(* IEC 61131-3 sources: brOscatLib/oscatBuild, 60 files *)

(* ---- oscatBuild.typ ---- *)
TYPE
END_TYPE

(* ---- AIR_DENSITY.st ---- *)
FUNCTION AIR_DENSITY
    (*http://www.oscat.de/images/OSCATBasic/oscat_basic333_en.pdf#page=426*)
    AIR_DENSITY := cPN * (1.0 - RH * SDD(T, TRUE) * RX / P) / (RL * ( T - cT0));

    (* original code used for rev 1.0

    SDD := SDD(T,FALSE);
    RF := RL / (1- RH*SDD/P*RX);
    AIR_DENSITY := P / (RF * (T-TK));

    *)

    (* revision history

    hm	29.10.2007	rev 1.0
    	original version

    hm	4.12.2007		rev 1.1
    	changed code for better performance

    hm	18. oct. 2008	rev 1.2
    	using phys constants

    hm	13. mar. 2009	rev 1.3
    	real constants updated to new systax using dot

    *)

END_FUNCTION

(* ---- AIR_ENTHALPY.st ---- *)
FUNCTION AIR_ENTHALPY
    (*http://www.oscat.de/images/OSCATBasic/oscat_basic333_en.pdf#page=427*)
    AIR_ENTHALPY := CPL * T + (CW * T + LH) * DEW_CON(RH,T);

    (* revision history

    hm	31.10.2007	rev 1.0
    	original version

    hm	2.11.2007		rev 1.1
    	deleted unused variable RF

    hm	2.12.2007		rev 1.2
    	changed code for better performance
    *)

END_FUNCTION

(* ---- BUILDING_VERSION.st ---- *)
FUNCTION BUILDING_VERSION
    (*http://www.oscat.de/images/OSCATBuilding/oscat_building100_en.pdf#page=11*)
    IF IN THEN
    	BUILDING_VERSION := DATE_TO_DWORD(D#2011-02-3);
    ELSE
    	BUILDING_VERSION := 100;
    END_IF

    (* revision history
    hm	6. oct 2006	rev 1.0
    	original version

    hm	16. dec 2007	rev 1.1
    	added possibility to return date and version depending on IN.

    *)
END_FUNCTION

(* ---- DEW_CON.st ---- *)
FUNCTION DEW_CON
    (*http://www.oscat.de/images/OSCATBasic/oscat_basic333_en.pdf#page=434*)
    (*	this code is good to read but need to be improoved
    	SDD := 6.1078*EXPT(10,(a*T)/(b+T));
    	DD := RH/100 * SDD;
    	V := LOG(DD/6.1078);
    	TD := b*V/(a-v);
    	DEW_CON := 0.1 * mw / RU * DD / (T - TK);
    *)
    IF RH > 0.0 AND T > -50.0 THEN
    	DEW_CON := 2.166824303E-2 * RH * SDD(T,FALSE)  / (T - cT0);
    ELSE
    	DEW_CON := 0.0;
    END_IF

    (*
    Bezeichnungen:
    r = relative Luftfeuchte
    T = Temperatur in °C
    TK = Temperatur in Kelvin (TK = T + 273.15)
    TD = Taupunkttemperatur in °C
    DD = Dampfdruck in hPa
    SDD = Sättigungsdampfdruck in hPa

    Parameter:
    a = 7.5, b = 237.3 für T >= 0
    a = 7.6, b = 240.7 für T < 0 über Wasser (Taupunkt)
    a = 9.5, b = 265.5 für T < 0 über Eis (Frostpunkt)

    R* = 8314.3 J/(kmol*K) (universelle Gaskonstante)
    mw = 18.016 kg (Molekulargewicht des Wasserdampfes)
    AF = absolute Feuchte in g Wasserdampf pro m3 Luft

    Formeln:

       1. SDD(T) = 6.1078 * 10((a*T)/(b+T))
       2. DD(r,T) = r/100 * SDD(T)
       3. r(T,TD) = 100 * SDD(TD) / SDD(T)
       4. TD(r,T) = b*v/(a-v) mit v(r,T) = log10(DD(r,T)/6.1078)
       5. AF(r,TK) = 105 * mw/R* * DD(r,T)/TK; AF(TD,TK) = 105 * mw/R* * SDD(TD)/TK

    *)

    (* revision history

    hm 29 apr 2007	rev 1.0
    	original version

    hm	13.sep 2007	rev 1.1
    	improoved coding for speed
    	deleted unused variabled SDD,DD,V, TD

    hm	2. dec 2007	rev 1.2
    	changed code for better performance
    	output is now in Gramms / Qubic meter

    hm	14. oct. 2008	rev 1.3
    	performance improvement

    hm	18. oct. 2008	rev 1.4
    	using phys constants

    hm	13. mar. 2009	rev 1.5
    	improved code

    hm	19. jan. 2011	rev 1.6
    	return value 0.0 if RH <= 0.0

    *)
END_FUNCTION

(* ---- DEW_RH.st ---- *)
FUNCTION DEW_RH
    (*http://www.oscat.de/images/OSCATBasic/oscat_basic333_en.pdf#page=435*)
    DEW_RH := LIMIT(0.0, VC / DEW_CON(1.0, T), 100.0);

    (* code before rev 1.1
    DEW_RH := VC / dew_con(100,T) * 100;
    IF DEW_RH > 100 THEN DEW_RH := 100; END_IF
    *)

    (* revision history
    hm	29. apr 2007	rev 1.0
    	original version

    hm	2. 12. 2007	rev 1.1
    	new code for better performance

    hm	13. mar. 2009	rev 1.2
    	real constants updated to new systax using dot

    *)
END_FUNCTION

(* ---- DEW_TEMP.st ---- *)
FUNCTION DEW_TEMP
    (*http://www.oscat.de/images/OSCATBasic/oscat_basic333_en.pdf#page=436*)
    IF RH > 0.0 THEN
    (*	old code was rewritten for better performance
    	SDD := 6.1078*EXPT(10,(a*T)/(b+T));
    	DD := RH/100 * SDD;
    	V := LOG(DD/6.1078);
    	DEW_TEMP := b*V/(a-V);
    *)
    	V := LOG(RH * 0.01 * EXP10((a*T) / (b+T)));
    	DEW_TEMP := b*V / (a-V);
    ELSE
    	DEW_TEMP:= cT0;
    END_IF

    (* revision history

    hm		2.10.2006	rev 1.0
    	original version created

    hm		29.4.2007	rev 1.1
    	checked for RH not to be 0 because log(0) is not defined

    hm		13.9.2007	rev 1.2
    	code rewritten for better performance

    hm	2. dec 2007	rev 1.3
    	changed code for better performance

    hm	8. jan 2008	rev 1.4
    	further improvement in performance

    hm	18. oct. 2008	rev 1.5
    	using phys constants

    hm	13. mar. 2009	rev 1.6
    	real constants updated to new systax using dot
    	function will now return -273.15 °C for RH = 0
    *)

    (*
    Bezeichnungen:
    r = relative Luftfeuchte
    T = Temperatur in °C
    TK = Temperatur in Kelvin (TK = T + 273.15)
    TD = Taupunkttemperatur in °C
    DD = Dampfdruck in hPa
    SDD = Sättigungsdampfdruck in hPa

    Parameter:
    a = 7.5, b = 237.3 für T >= 0
    a = 7.6, b = 240.7 für T < 0 über Wasser (Taupunkt)
    a = 9.5, b = 265.5 für T < 0 über Eis (Frostpunkt)

    R* = 8314.3 J/(kmol*K) (universelle Gaskonstante)
    mw = 18.016 kg (Molekulargewicht des Wasserdampfes)
    AF = absolute Feuchte in g Wasserdampf pro m3 Luft

    Formeln:

       1. SDD(T) = 6.1078 * 10((a*T)/(b+T))
       2. DD(r,T) = r/100 * SDD(T)
       3. r(T,TD) = 100 * SDD(TD) / SDD(T)
       4. TD(r,T) = b*V/(a-V) mit V(r,T) = log10(DD(r,T)/6.1078)
       5. AF(r,TK) = 105 * mw/R* * DD(r,T)/TK; AF(TD,TK) = 105 * mw/R* * SDD(TD)/TK

    *)
END_FUNCTION

(* ---- HEAT_INDEX.st ---- *)
FUNCTION HEAT_INDEX
    (*http://www.oscat.de/images/OSCATBasic/oscat_basic333_en.pdf#page=436*)
    IF RH < 20.0 OR T < 20.0 THEN
    	HEAT_INDEX := T;
    ELSE
    	RH2 := RH * RH;
    	T := C_TO_F(T);
    	T2 := T * T;
    	HEAT_INDEX := -42.379 + 2.04901523 * T - 6.83783E-3 * T2
    			+ RH * (10.1433127 - 0.22475541 * T + 1.22874E-3 * T2)
    			+ RH2 * (8.5282E-4 * T - 5.481717E-2 - 1.99E-6 * T2);
    	HEAT_INDEX := F_TO_C(HEAT_INDEX);
    END_IF

    (* revision history

    hm 27.2.2007		rev 1.1
    	deleted unused variables rh3 and T3

    hm	2.12.2007		rev 1.2
    	changed code for better performance

    hm	13. mar. 2009	rev 1.3
    	real constants updated to new systax using dot

    *)
END_FUNCTION

(* ---- SDD.st ---- *)
FUNCTION SDD
    (*http://www.oscat.de/images/OSCATBasic/oscat_basic333_en.pdf#page=445*)
    IF ICE THEN
    	SDD := 611.153 * EXP(22.4433 * T / (272.186 + T));
    ELSE
    	SDD := 611.213 * EXP(17.5043 * T / (241.2 + T));
    END_IF

    (* revision history

    hm 29 oct 2007		rev 1.0
    	original version

    hm	2. dec 2007		rev 1.1
    	changed code for better performance
    *)
END_FUNCTION

(* ---- SDD_NH3.st ---- *)
FUNCTION SDD_NH3
    (*http://www.oscat.de/images/OSCATBasic/oscat_basic333_en.pdf#page=446*)
    (*
    calculate according to NIST
    Antoine Equation Parameters
    log10(P) = A - (B / (T + C))
    	P = vapor pressure (bar)
    	T = temperature (K)
    Temperature (K)	A	B	C	Reference	Comment

     T = 164.0 - 239.5, A =	3.18757, B =506.713, C=-80.78	Stull, 1947	Coefficents calculated by NIST from author's data.
     T = 239.5 - 371.4, A =	4.86886, B = 1113.928, C = -10.409	Stull, 1947	Coefficents calculated by NIST from author's data.
    *)

    IF T < -33.65 THEN
    	SDD_NH3 := EXP(7.3396511649 - ( 1166.7498002 / ( T + 192.37 )));
    ELSE
    	SDD_NH3 := EXP(11.210964456 - ( 2564.9140075 / ( T + 262.741 )));
    END_IF

    (* revision history

    hm 19 aug 2009		rev 1.0
    	original version

    *)
END_FUNCTION

(* ---- SDT_NH3.st ---- *)
FUNCTION SDT_NH3
    (*http://www.oscat.de/images/OSCATBasic/oscat_basic333_en.pdf#page=446*)
    (*
    calculate according to NIST
    Antoine Equation Parameters
    log10(P) = A - (B / (T + C))
    	P = vapor pressure (bar)
    	T = temperature (K)
    Temperature (K)	A	B	C	Reference	Comment

     T = 164.0 - 239.5, A =	3.18757, B =506.713, C=-80.78	Stull, 1947	Coefficents calculated by NIST from author's data.
     T = 239.5 - 371.4, A =	4.86886, B = 1113.928, C = -10.409	Stull, 1947	Coefficents calculated by NIST from author's data.
    *)

    IF P < 1.0E-3 THEN
    	SDT_NH3 := -110.0;
    ELSIF P < 1.0 THEN
    	SDT_NH3 := 506.713 / (3.18757 - LOG(P)) - 192.37 ;
    ELSE
    	SDT_NH3 := 1113.928 / (4.86886 - LOG(P)) - 262.71 ;
    END_IF

    (* revision history

    hm 20 aug 2009		rev 1.0
    	original version

    *)
END_FUNCTION

(* ---- TANK_VOL1.st ---- *)
FUNCTION TANK_VOL1
    (*http://www.oscat.de/images/OSCATBasic/oscat_basic333_en.pdf#page=448*)
    TANK_VOL1 := CIRCLE_SEG(TR, H) * TL;

    (* revision histroy
    hm	10. mar 2010	rev 1.0
    	original version

    *)
END_FUNCTION

(* ---- TANK_VOL2.st ---- *)
FUNCTION TANK_VOL2
    (*http://www.oscat.de/images/OSCATBasic/oscat_basic333_en.pdf#page=448*)
    TANK_VOL2 := cPI * H * H * (TR - H/3.0);

    (* revision histroy
    hm	10. mar 2010	rev 1.0
    	original version

    *)
END_FUNCTION

(* ---- TIMER_EVENT_DECODE.st ---- *)
FUNCTION TIMER_EVENT_DECODE
    (*http://www.oscat.de/images/OSCATBuilding/oscat_building100_en.pdf#page=62*)
    (* a timer EVENT is specified as follows:
    	$typ;ch;day;start;duration;land;lor#
    $ 		= start of definition
    typ 	= type of definition	(number)
    channel	= channel number		(number)
    day 	= day number			(number)
    start	= start time			(time of day)
    duration= duration of EVENT		(time)
    land	= mask for output AND	(8bit value)
    lor		= mask for ourput OR	(8bit value)
    #		= end of definition
    *)

    (* check for start and ending character *)
    IF (LEFT(EVENT,1) <> '<') AND (RIGHT(EVENT,1) <> '>') THEN RETURN; END_IF
    stop := LEN(EVENT);
    pt := ADR(EVENT);
    start := 2;

    (* parse the string for next ; *)
    FOR pos := 2 TO stop DO
    	IF pt[pos] = 59 OR pt[pos] = 62 THEN
    		tmp := MID(EVENT, pos - start, start);
    		CASE step OF
    			0:	(* read type *)
    				TIMER_EVENT_DECODE.typ := FSTRING_TO_BYTE(tmp);

    			1:	(* read channel *)
    				TIMER_EVENT_DECODE.channel := FSTRING_TO_BYTE(tmp);

    			2:	(* read day *)
    				IF IS_CC(tmp,'0123456789abcdefABCDEF#') THEN
    					TIMER_EVENT_DECODE.day := FSTRING_TO_BYTE(tmp);
    				ELSIF TIMER_EVENT_DECODE.typ = 2 THEN
    					TIMER_EVENT_DECODE.DAY := FSTRING_TO_WEEK(tmp, LANG);
    				ELSE
    					TIMER_EVENT_DECODE.DAY := INT_TO_BYTE(FSTRING_TO_WEEKDAY(tmp, LANG));
    				END_IF

    			3:	(* read start *)
    				TIMER_EVENT_DECODE.start := STRING_TO_TOD(tmp);

    			4:	(* read duaration *)
    				TIMER_EVENT_DECODE.duration := STRING_TO_TIME(tmp);

    			5:	(* read land *)
    				TIMER_EVENT_DECODE.land := FSTRING_TO_BYTE(tmp);

    			6:	(* read lor *)
    				TIMER_EVENT_DECODE.LOR := FSTRING_TO_BYTE(tmp);
    		END_CASE
    		start := pos + 1;
    		step := step + 1;
    	END_IF
    END_FOR

    (* revision history
    hm	17. jun 2008	rev 1.0
    	original version

    hm	25. oct. 2008	rev 1.1
    	adding input LANG for language selection
    *)

END_FUNCTION

(* ---- WATER_CP.st ---- *)
FUNCTION WATER_CP
    (*http://www.oscat.de/images/OSCATBasic/oscat_basic333_en.pdf#page=452*)
    WATER_CP := LINEAR_INT(T, data, Pts);

    (*
        °C - die Celsius-Temperatur in Grad Celsius
        v – das spezifische Volumen in Kubikdezimeter je Kilogramm dm³/kg
        h – die spezifische Enthalpie in Kilojoule je Kilogramm 	kJ/kg
        u – die spezifische Innere Energie in Kilojoule je Kilogramm 	kJ/kg
        s – die spezifische Entropie in Kilojoule je Kilogramm mal Kelvin 	kJ/(kg·K)
        cp - die spezifische Wärmekapazität bei konstantem Druck in Kilojoule je Kilogramm mal Kelvin 	kJ/(kg·K)
        Y – Volumenausdehnungskoeffizient in 10-3 durch Kelvin  10-3/K
        L – Wärmeleitfähigkeit in Milliwatt je Meter mal Kelvin  mW / (m·K)
        n – Viskosität in Mikropascal mal Sekunde uPa·s
        s ? – Oberflächenspannung in Millinewton je Meter  mN/m

    °C 		v 				h 			u 		s 			cp 		Y 		L		n		s
    -20		1,006580
    0 		1,000160 		0,06 		-0,04 	-0,0001 	4,228 	-0,080 	561,0 	1792 	75,65
    4		1,000028
    5 		1,0000 		21,1 		21,0 	0,076 		4,200 	0,011 	570,6 	1518 	74,95
    10 		1,0003 		42,1 		42,0 	0,151 		4,188 	0,087 	580,0 	1306 	74,22
    15 		1,0009 		63,0 		62,9 	0,224 		4,184 	0,152 	589,4 	1137 	73,49
    20 		1,001797 		83,9 		83,8 	0,296 		4,183 	0,209 	598,4 	1001 	72,74
    25 		1,0029 		104,8 		104,7 	0,367 		4,183 	0,259 	607,2 	890,4 	71,98
    30 		1,0044 		125,8 		125,7 	0,437 		4,183 	0,305 	615,5 	797,7 	71,20
    35 		1,0060 		146,7 		146,6 	0,505 		4,183 	0,347 	623,3 	719,6 	70,41
    40 		1,007842 		167,58 	167,5 	0,572 		4,182 	0,386 	630,6 	653,3 	69,60
    45 		1,0099 		188,5 		188,4 	0,638 		4,182 	0,423 	637,3 	596,3 	68,78
    50 		1,0121 		209,4 		209,3 	0,704 		4,181 	0,457 	643,6 	547,1 	67,95
    60 		1,017089 		251,2 		251,1 	0,831 		4,183 	0,522 	654,4 	466,6 	66,24
    70 		1,0227 		293,1 		293,0 	0,955 		4,187 	0,583 	663,1 	404,1 	64,49
    80 		1,029027 		335,0 		334,9 	1,075 		4,194 	0,640 	670,0 	354,5 	62,68
    90 		1,0359 		377,0 		376,9 	1,193 		4,204 	0,696 	675,3 	314,6 	60,82
    99,63 	1,0431 		417,5 		417,4 	1,303 		4,217 	0,748 	679,0 	283,0 	58,99
    100	1,043453		419,1

    Stoffdaten von Wasser Quelle Wickipedia

    Wasser hat unter Normaldruck seine größte Dichte von 1000 Kilogramm pro Kubikmeter bei 3,98 °C und zeigt damit eine Dichteanomalie.
    Diese besteht darin, dass sich Wasser unterhalb von 3,98 °C bei weiterer Temperaturverringerung, auch beim Wechsel zum festen
    Aggregatzustand, wieder ausdehnt, was man nur von wenigen Stoffen kennt. Die derzeit genauesten publizierten Werte für die maximale
    Dichte liegen bei (999,974950 ± 0,00084) kg/m³ und bei (3,983 ± 0,00067) °C für die Temperatur, bei der dieser Wert erreicht wird.
    Die Werte stellen einen Mittelwert der von verschiedenen physikalischen Instituten veröffentlichten Zahlen dar (Stand 2001).

    Die Berechnung der Dichte von luftfreiem Wasser DLF in Abhängigkeit von der Temperatur T ([T] = °C) kann mit Hilfe der folgenden
    Virialgleichung erfolgen:
    : \frac{D_{\rm LF}}{\rm g/l} = \frac{a_0 + a_1 T + a_2 T2 + a_3 T3 + a_4 T4 + a_5 T5}{1 + b T}.
    mit den Koeffizienten: a0 = 999,83952; a1 = 16,952577 (°C)-1; a2 = -7,9905127·10-3 (°C)-2; a3 = -4,6241757·10-5 (°C)-3;
    a4 = 1,0584601·10-7 (°C)-4; a5 = -2,8103006·10-10 (°C)-5 und b = 0,0168872.
    Für die Berechnung der Dichte von luftgesättigtem Wasser korrigiert man den Wert nach
    DLG/(g/l) = DLF/(g/l) - 0,004612 + 0,000106 (°C)-1·T. (Quelle: PTB-Mitteilungen 100/3-90)

    *)

    (* revision history

    hm	29.10.2007	rev 1.0
    	original version

    hm	27. dec 2007	rev 1.1
    	increased accuracy

    hm	13. mar. 2009	rev 1.2
    	real constants updated to new systax using dot

    *)

END_FUNCTION

(* ---- WATER_DENSITY.st ---- *)
FUNCTION WATER_DENSITY
    (*http://www.oscat.de/images/OSCATBasic/oscat_basic333_en.pdf#page=452*)
    T2 := T * T;
    T4 := T2 * T2;
    WATER_DENSITY := (a0 + a1*T + a2*T2 + a3*T2*T + a4*T4 + a5*T4*T) / (1.0 + b*T);
    IF SAT THEN WATER_DENSITY := WATER_DENSITY - 0.004612 + 0.000106 * T; END_IF

    (* revision history

    hm	13.9.2007		rev 1.0
    	original version

    hm	2.12.2007		rev 1.1
    	changed code for better performance

    hm	13. mar. 2009	rev 1.2
    	real constants updated to new systax using dot

    *)

    (*
        °C - die Celsius-Temperatur in Grad Celsius
        v – das spezifische Volumen in Kubikdezimeter je Kilogramm dm³/kg
        h – die spezifische Enthalpie in Kilojoule je Kilogramm 	kJ/kg
        u – die spezifische Innere Energie in Kilojoule je Kilogramm 	kJ/kg
        s – die spezifische Entropie in Kilojoule je Kilogramm mal Kelvin 	kJ/(kg·K)
        cp - die spezifische Wärmekapazität bei konstantem Druck in Kilojoule je Kilogramm mal Kelvin 	kJ/(kg·K)
        Y – Volumenausdehnungskoeffizient in 10-3 durch Kelvin  10-3/K
        L – Wärmeleitfähigkeit in Milliwatt je Meter mal Kelvin  mW / (m·K)
        n – Viskosität in Mikropascal mal Sekunde uPa·s
        s ? – Oberflächenspannung in Millinewton je Meter  mN/m

    °C 		v 				h 			u 		s 			cp 		Y 		L		n		s
    -20		1,006580
    0 		1,000160 		0,06 		-0,04 	-0,0001 	4,228 	-0,080 	561,0 	1792 	75,65
    4		1,000028
    5 		1,0000 		21,1 		21,0 	0,076 		4,200 	0,011 	570,6 	1518 	74,95
    10 		1,0003 		42,1 		42,0 	0,151 		4,188 	0,087 	580,0 	1306 	74,22
    15 		1,0009 		63,0 		62,9 	0,224 		4,184 	0,152 	589,4 	1137 	73,49
    20 		1,001797 		83,9 		83,8 	0,296 		4,183 	0,209 	598,4 	1001 	72,74
    25 		1,0029 		104,8 		104,7 	0,367 		4,183 	0,259 	607,2 	890,4 	71,98
    30 		1,0044 		125,8 		125,7 	0,437 		4,183 	0,305 	615,5 	797,7 	71,20
    35 		1,0060 		146,7 		146,6 	0,505 		4,183 	0,347 	623,3 	719,6 	70,41
    40 		1,007842 		167,58 	167,5 	0,572 		4,182 	0,386 	630,6 	653,3 	69,60
    45 		1,0099 		188,5 		188,4 	0,638 		4,182 	0,423 	637,3 	596,3 	68,78
    50 		1,0121 		209,4 		209,3 	0,704 		4,181 	0,457 	643,6 	547,1 	67,95
    60 		1,017089 		251,2 		251,1 	0,831 		4,183 	0,522 	654,4 	466,6 	66,24
    70 		1,0227 		293,1 		293,0 	0,955 		4,187 	0,583 	663,1 	404,1 	64,49
    80 		1,029027 		335,0 		334,9 	1,075 		4,194 	0,640 	670,0 	354,5 	62,68
    90 		1,0359 		377,0 		376,9 	1,193 		4,204 	0,696 	675,3 	314,6 	60,82
    99,63 	1,0431 		417,5 		417,4 	1,303 		4,217 	0,748 	679,0 	283,0 	58,99
    100	1,043453		419,1

    Stoffdaten von Wasser Quelle Wickipedia

    *)

END_FUNCTION

(* ---- WATER_ENTHALPY.st ---- *)
FUNCTION WATER_ENTHALPY
    (*http://www.oscat.de/images/OSCATBasic/oscat_basic333_en.pdf#page=453*)
    WATER_ENTHALPY := LINEAR_INT(T, data, Pts);

    (*
        °C - die Celsius-Temperatur in Grad Celsius
        v – das spezifische Volumen in Kubikdezimeter je Kilogramm dm³/kg
        h – die spezifische Enthalpie in Kilojoule je Kilogramm 	kJ/kg
        u – die spezifische Innere Energie in Kilojoule je Kilogramm 	kJ/kg
        s – die spezifische Entropie in Kilojoule je Kilogramm mal Kelvin 	kJ/(kg·K)
        cp - die spezifische Wärmekapazität bei konstantem Druck in Kilojoule je Kilogramm mal Kelvin 	kJ/(kg·K)
        Y – Volumenausdehnungskoeffizient in 10-3 durch Kelvin  10-3/K
        L – Wärmeleitfähigkeit in Milliwatt je Meter mal Kelvin  mW / (m·K)
        n – Viskosität in Mikropascal mal Sekunde uPa·s
        s ? – Oberflächenspannung in Millinewton je Meter  mN/m

    °C 		v 				h 			u 		s 			cp 		Y 		L		n		s
    -20		1,006580
    0 		1,000160 		0,06 		-0,04 	-0,0001 	4,228 	-0,080 	561,0 	1792 	75,65
    4		1,000028
    5 		1,0000 		21,1 		21,0 	0,076 		4,200 	0,011 	570,6 	1518 	74,95
    10 		1,0003 		42,1 		42,0 	0,151 		4,188 	0,087 	580,0 	1306 	74,22
    15 		1,0009 		63,0 		62,9 	0,224 		4,184 	0,152 	589,4 	1137 	73,49
    20 		1,001797 		83,9 		83,8 	0,296 		4,183 	0,209 	598,4 	1001 	72,74
    25 		1,0029 		104,8 		104,7 	0,367 		4,183 	0,259 	607,2 	890,4 	71,98
    30 		1,0044 		125,8 		125,7 	0,437 		4,183 	0,305 	615,5 	797,7 	71,20
    35 		1,0060 		146,7 		146,6 	0,505 		4,183 	0,347 	623,3 	719,6 	70,41
    40 		1,007842 		167,58 	167,5 	0,572 		4,182 	0,386 	630,6 	653,3 	69,60
    45 		1,0099 		188,5 		188,4 	0,638 		4,182 	0,423 	637,3 	596,3 	68,78
    50 		1,0121 		209,4 		209,3 	0,704 		4,181 	0,457 	643,6 	547,1 	67,95
    60 		1,017089 		251,2 		251,1 	0,831 		4,183 	0,522 	654,4 	466,6 	66,24
    70 		1,0227 		293,1 		293,0 	0,955 		4,187 	0,583 	663,1 	404,1 	64,49
    80 		1,029027 		335,0 		334,9 	1,075 		4,194 	0,640 	670,0 	354,5 	62,68
    90 		1,0359 		377,0 		376,9 	1,193 		4,204 	0,696 	675,3 	314,6 	60,82
    99,63 	1,0431 		417,5 		417,4 	1,303 		4,217 	0,748 	679,0 	283,0 	58,99
    100	1,043453		419,1

    Stoffdaten von Wasser Quelle Wickipedia

    Wasser hat unter Normaldruck seine größte Dichte von 1000 Kilogramm pro Kubikmeter bei 3,98 °C und zeigt damit eine Dichteanomalie.
    Diese besteht darin, dass sich Wasser unterhalb von 3,98 °C bei weiterer Temperaturverringerung, auch beim Wechsel zum festen
    Aggregatzustand, wieder ausdehnt, was man nur von wenigen Stoffen kennt. Die derzeit genauesten publizierten Werte für die maximale
    Dichte liegen bei (999,974950 ± 0,00084) kg/m³ und bei (3,983 ± 0,00067) °C für die Temperatur, bei der dieser Wert erreicht wird.
    Die Werte stellen einen Mittelwert der von verschiedenen physikalischen Instituten veröffentlichten Zahlen dar (Stand 2001).

    Die Berechnung der Dichte von luftfreiem Wasser DLF in Abhängigkeit von der Temperatur T ([T] = °C) kann mit Hilfe der folgenden
    Virialgleichung erfolgen:
    : \frac{D_{\rm LF}}{\rm g/l} = \frac{a_0 + a_1 T + a_2 T2 + a_3 T3 + a_4 T4 + a_5 T5}{1 + b T}.
    mit den Koeffizienten: a0 = 999,83952; a1 = 16,952577 (°C)-1; a2 = -7,9905127·10-3 (°C)-2; a3 = -4,6241757·10-5 (°C)-3;
    a4 = 1,0584601·10-7 (°C)-4; a5 = -2,8103006·10-10 (°C)-5 und b = 0,0168872.
    Für die Berechnung der Dichte von luftgesättigtem Wasser korrigiert man den Wert nach
    DLG/(g/l) = DLF/(g/l) - 0,004612 + 0,000106 (°C)-1·T. (Quelle: PTB-Mitteilungen 100/3-90)

    *)

    (* revision history
    hm	13. mar. 2009	rev 1.0
    	original version

    hm	13. mar. 2009	rev 1.1
    	real constants updated to new systax using dot

    *)
END_FUNCTION

(* ---- WCT.st ---- *)
FUNCTION WCT
    (*http://www.oscat.de/images/OSCATBasic/oscat_basic333_en.pdf#page=453*)
    IF V < 5.0 OR T > 10.0 THEN
    	WCT := T;
    ELSE
    	WCT := 13.12 + 0.6215 * T +(0.3965 * T - 11.37) * EXP(LN(V) * 0.16);
    END_IF

    (* revision history
    hm	7 feb 2007		rev 1.0
    	original version

    hm	7 dec 2007	rev 1.1
    	changed code for better performance

    hm	13. mar. 2009	rev 1.2
    	real constants updated to new systax using dot

    *)
END_FUNCTION

(* ---- ACTUATOR_2P.st ---- *)
FUNCTION_BLOCK ACTUATOR_2P
    (*http://www.oscat.de/images/OSCATBuilding/oscat_building100_en.pdf#page=12*)
    (* run the autorun timer *)
    timer(trun := SELF_ACT_PULSE * (2 * SELF_ACT_CYCLES), toff := SELF_ACT_TIME, TEST := TEST, ARE := ARE, ARX := ARX);
    ARO := timer.ARO;

    (* run the pulse width generator *)
    IF ARO THEN
    	pwgen(PTL := SELF_ACT_PULSE, PTH := SELF_ACT_PULSE);
    	OUT := pwgen.Q;
    ELSIF IN < SENS THEN
    	OUT := FALSE;
    ELSIF IN > BYTE#255 - SENS THEN
    	OUT := TRUE;
    ELSE
    	pwgen.PTH := (CYCLE_TIME * BAND_B(IN,SENS)) / 255;
    	pwgen.PTL := CYCLE_TIME - pwgen.PTH;
    	pwgen();
    	OUT := pwgen.Q;
    END_IF

    (* revision history
    hm	7.10.2006 		rev 1.1
    	changed error pos could not reach 1 or 0 under certain conditions due to error IN code.
    	changed on and off IN force and force_in for better usability.

    hm	17.1.2007		rev 1.2
    	deleted unused variable time_overflow

    hm	15.9.2007		rev 1.3
    	replaced time() with T_PLC_MS for compatibility and performance reasons

    hm	19. 11 2007		rev 1.4
    	replaced left over statement time() with tx

    hm	27. 12. 2007	REV 1.5
    	CHANGED CODE FOR BETTER PERFORMANCE

    hm	21. oct. 2008	rev 1.6
    	code optimized

    hm	23. nov. 2008	rev 2.0
    	new code using library modules

    hm	24. jan. 2009	rev 2.1
    	deleted unused var inb
    *)
END_FUNCTION_BLOCK

(* ---- ACTUATOR_3P.st ---- *)
FUNCTION_BLOCK ACTUATOR_3P
    (*http://www.oscat.de/images/OSCATBuilding/oscat_building100_en.pdf#page=13*)
    (* read system timer *)
    tx := DWORD_TO_TIME(T_PLC_MS());

    (* check TEST input *)
    IF TEST THEN
    	STATUS := 103;
    	start := tx;
    	ARX := TRUE;
    END_IF

    CASE STATUS OF
    	0:	(* power on setup *)
    		IF ARE AND NOT ARX THEN
    			STATUS := 103;
    			start := tx;
    			ARX := TRUE;
    		END_IF

    	100:	(* normal operation *)
    		(* check for auto diagnostics *)
    		IF T_DIAG > T#0s AND tx > next_diag AND ARE AND NOT ARX THEN
    				STATUS := 103;
    				start := tx;
    				ARX := TRUE;

    		(* check for auto calibration *)
    		ELSIF T_CAL > T#0s AND tx > next_cal AND ARE AND NOT ARX THEN
    			IF POS > BYTE#127 THEN
    				OUT1 := TRUE;
    				OUT2 := FALSE;
    				ramp.IN := 255;
    				ARX := TRUE;
    			ELSE
    				OUT1 := FALSE;
    				OUT2 := TRUE;
    				ramp.IN := 0;
    				ARX := TRUE;
    			END_IF
    			STATUS := 101;
    			start := tx;
    		ELSE
    			(* increment next_cal if not active *)
    			IF NOT(OUT1 OR OUT2) THEN next_cal := next_cal + (tx-last); END_IF
    			(* set ramp generator to IN *)
    			ramp.IN := IN;
    		END_IF

    	101:	(* calibrate *)
    		IF tx - start < T_EXT THEN
    			next_cal := tx + T_CAL;
    		ELSIF SWITCH_AVAIL AND END_POS THEN
    			STATUS := 100;
    			ARX := FALSE;
    		ELSIF tx - start > T_EXT + T_RUN THEN
    			ERROR := SWITCH_AVAIL;
    			ARX := FALSE;
    		END_IF

    	103:	(* diagnostics up*)
    		(* run up for T_EXT *)
    		IF tx - start < T_EXT THEN
    			ERROR := FALSE;
    			ramp.TR := T_RUN;
    			ramp.TF := T_RUN;
    			OUT1 := TRUE;
    			OUT2 := FALSE;
    			ramp.IN := 255;
    		ELSIF SWITCH_AVAIL AND END_POS THEN
    			ramp.TR := tx - start;
    			STATUS := 104;
    		ELSIF tx - start > T_EXT + T_RUN THEN
    			ERROR := SWITCH_AVAIL;
    			STATUS := 104;
    			start := tx;
    		END_IF

    	104:	(* diagnostics dn*)
    		IF tx - start < T_EXT THEN
    			OUT1 := FALSE;
    			OUT2 := TRUE;
    			ramp.IN := 0;
    			next_diag := tx + T_DIAG;
    		ELSIF SWITCH_AVAIL AND END_POS THEN
    			ramp.TR := tx - start;
    			(* check if runtimes differ by more than 10% *)
    			IF DINT_TO_TIME(ABS(TIME_TO_DINT(ramp.TR) - TIME_TO_DINT(ramp.TF))*10) > T_RUN THEN ERROR := TRUE; END_IF
    			STATUS := 100;
    			ARX := FALSE;
    			next_cal := tx + T_CAL;
    		ELSIF tx - start > T_EXT + T_RUN THEN
    			IF SWITCH_AVAIL THEN ERROR := TRUE; END_IF
    			STATUS := 100;
    			ARX := FALSE;
    			next_cal := tx + T_CAL;
    		END_IF
    END_CASE

    (* internal flap simulation and output activation *)
    ramp(OUT := POS);
    IF STATUS = 100 THEN
    	OUT1 := ramp.UP;
    	OUT2 := ramp.DN;
    END_IF

    (* adjust position if end switch is active *)
    IF SWITCH_AVAIL AND END_POS THEN
    	POS := SEL(POS > 127, 0, 255);
    	next_cal := tx + T_CAL;
    END_IF

    (* set last to tx for next cycle *)
    last := tx;

    (* revision history

    hm	19. oct 2006	rev 1.1
    	added security checks for end_switch to avoid overrun of the end_switch, hans

    hm	23. jan 2007	rev 1.2
    	deleted unused variables force_on and force_off

    hm	15. sep 2007	 rev 1.3
    	replaced Time() with T_PLC_MS for compatibility and performance reasons

    hm	28. jan 2010	rev 2.0
    	new code and new features

    *)

END_FUNCTION_BLOCK

(* ---- ACTUATOR_A.st ---- *)
FUNCTION_BLOCK ACTUATOR_A
    (*http://www.oscat.de/images/OSCATBuilding/oscat_building100_en.pdf#page=15*)
    (* run the system timer, if SELF_ACT_TIME = t#0s then state IS set to 0 *)
    timer(T0 := RUNTIME, T1 := RUNTIME, T3 := SELF_ACT_TIME, sl := DX AND NOT dx_edge, sx := 0, S0 := SELF_ACT_TIME > t#0s);
    dx_edge := DX;

    CASE timer.STATE OF
    	0: 	(* self act min value *)
    		Y := OUT_MIN;
    	1:	(* self_act max value *)
    		Y := OUT_MAX;
    	3:	(* normal operation *)
    		IF RV THEN
    			Y := OUT_MAX - (OUT_MAX - OUT_MIN) * SEL(IS, I1, I2) / 255;
    		ELSE
    			Y := (OUT_MAX - OUT_MIN) * SEL(IS, I1, I2) / 255 + OUT_MIN;
    		END_IF
    END_CASE

    (*
    hm 	8. nov. 2008	rev 1.0
    	original version

    *)
END_FUNCTION_BLOCK

(* ---- ACTUATOR_COIL.st ---- *)
FUNCTION_BLOCK ACTUATOR_COIL
    (*http://www.oscat.de/images/OSCATBuilding/oscat_building100_en.pdf#page=16*)
    (* read system time *)
    now := T_PLC_MS();

    (* initialize for first cycle *)
    IF NOT init THEN
    	last := now;
    	init := TRUE;
    ELSIF IN THEN
    	OUT := TRUE;
    	STATUS := 101; (* activated by input *)
    	last := now;
    ELSE
    	OUT := FALSE;
    	STATUS := 100; (* disabled *)
    	(* now we need to check for self activation *)
    	tx := now - last;
    	IF (SELF_ACT_CYCLE > T#0s) AND (tx >= TIME_TO_DWORD(SELF_ACT_CYCLE)) THEN
    		OUT := TRUE;
    		STATUS := 102; (* auto activation *)
    		IF tx >= TIME_TO_DWORD(SELF_ACT_CYCLE + SELF_ACT_TIME) THEN
    			last := now;
    			OUT := FALSE;
    			STATUS := 100; (* idle *)
    		END_IF
    	END_IF
    END_IF

    (*
    revision history:

    hm		1. jun. 2008 	rev 1.0
    	original version

    *)
END_FUNCTION_BLOCK

(* ---- ACTUATOR_PUMP.st ---- *)
FUNCTION_BLOCK ACTUATOR_PUMP
    (*http://www.oscat.de/images/OSCATBuilding/oscat_building100_en.pdf#page=16*)
    tx := DWORD_TO_TIME(T_PLC_MS());

    IF NOT init THEN
    	init := TRUE;
    	last_change := tx;
    ELSIF RST THEN
    	RST := FALSE;
    	RUNTIME := 0;
    	CYCLES := 0;
    ELSIF MANUAL AND NOT PUMP AND NOT old_man THEN
    	last_change := tx;
    	PUMP := TRUE;
    ELSIF NOT MANUAL AND old_man AND PUMP AND NOT IN THEN
    	last_change := tx;
    	PUMP := FALSE;
    ELSIF IN AND NOT PUMP AND tx - last_change >= MIN_OFFTIME THEN
    	last_change := tx;
    	PUMP := TRUE;
    ELSIF PUMP AND NOT IN AND NOT MANUAL AND tx - last_change >= MIN_ONTIME THEN
    	last_change := tx;
    	PUMP := FALSE;
    ELSIF NOT PUMP AND (tx - last_change >= RUN_EVERY) AND (RUN_EVERY > T#0s) THEN
    	last_change := tx;
    	PUMP := TRUE;
    END_IF

    meter(IN := PUMP, seconds := RUNTIME, CYCLES := CYCLES);
    old_man := MANUAL;

    (*
    hm	27.12.2006		rev 1.1
    	fixed a failure while the PUMP would run for tmin after startup.

    hm	15.9.2007		rev 1.2
    	replaced Time() with T_PLC_MS for compatibility and performance reasons

    hm	13. oct. 2008	rev 1.3
    	auto activation can now be disabled when RUN_EVERY = t#0s

    hm	21. oct. 2008	rev 1.4
    	changed to use ontime rev 2.0

    *)
END_FUNCTION_BLOCK

(* ---- ACTUATOR_UD.st ---- *)
FUNCTION_BLOCK ACTUATOR_UD
    (*http://www.oscat.de/images/OSCATBuilding/oscat_building100_en.pdf#page=17*)
    (* read system time *)
    tx := DWORD_TO_TIME(T_PLC_MS());

    IF NOT init THEN
    	(* INITIALIZATION AT FIRST CALL *)
    	last := tx;
    	init := TRUE;
    ELSIF OFF THEN
    	(* emergency shut OFF detected *)
    	YUP := FALSE;
    	YDN := FALSE;
    	last := tx;
    	STATUS := 101;

    (* Watch FOR MIN TON TIME *)
    ELSIF ((YUP OR YDN) AND tx - last < TON) THEN
    	RETURN;
    ELSIF NOT YUP AND NOT YDN AND tx - last < TOFF THEN
    	RETURN;

    (* MANUAL operation *)
    ELSIF MANUAL THEN
    	STATUS := 102;
    	(* directional chage set both outs 0 first *)
    	IF YUP AND NOT UP OR YDN AND NOT DN THEN
    		YDN := FALSE;
    		YUP := FALSE;
    		last := tx;
    	(* MANUAL UP operation *)
    	ELSIF UP AND NOT DN AND NOT OFF THEN
    		YDN := FALSE;
    		YUP := TRUE;
    		last := tx;
    		STATUS := 103;
    	(* MANUAL down operation *)
    	ELSIF DN AND NOT UP AND NOT OFF THEN
    		YUP := FALSE;
    		YDN := TRUE;
    		last := tx;
    		STATUS := 104;
    	(* maual mode but no UP or down *)
    	ELSE
    		IF YUP OR YDN THEN last := tx; END_IF
    		YUP := FALSE;
    		YDN := FALSE;
    	END_IF

    (* automatic operation *)
    ELSE
    	(* directional change set outputs low first *)
    	IF YUP AND NOT UD OR YDN AND UD THEN
    		YUP := FALSE;
    		YDN := FALSE;
    		last := tx;
    	(* automatic UP operation *)
    	ELSIF UD AND ON AND NOT OFF THEN
    		YDN := FALSE;
    		YUP := TRUE;
    		last := tx;
    		STATUS := 111;

    	(* automatic down operation *)
    	ELSIF NOT UD AND ON AND NOT OFF THEN
    		YUP := FALSE;
    		YDN := TRUE;
    		last := tx;
    		STATUS := 112;
    	(* standby mode *)
    	ELSE
    		IF YUP OR YDN THEN last := tx; END_IF
    		YUP := FALSE;
    		YDN := FALSE;
    		STATUS := 110;
    	END_IF
    END_IF

    (* make sure YUP and YDN are never ON at the same time *)
    IF YDN AND YUP_IN AND OUT_RETURN THEN
    	YDN := FALSE;
    	STATUS := 1;
    END_IF
    IF YUP AND YDN_IN AND OUT_RETURN THEN
    	YUP := FALSE;
    	STATUS := 2;
    END_IF

    (* revision history
    hm 22. jan 2007	rev 1.1
    	added STATUS output
    	changed inputs TON, TOFF to config variables
    	added config var OUT_RETURN to enable YUP_IN and YDN_IN
    	MANUAL mod will override automatic mode

    hm	15.9.2007	rev 1.2
    	replaced Time() with T_PLC_MS for compatibility and performance reasons

    hm	17. oct. 2008	rev 1.3
    	deleted unnecessary initialization with 0
    *)
END_FUNCTION_BLOCK

(* ---- AUTORUN.st ---- *)
FUNCTION_BLOCK AUTORUN
    (*http://www.oscat.de/images/OSCATBuilding/oscat_building100_en.pdf#page=19*)
    (* run the integrator when T_off > T#0s *)
    IF TOFF > T#0s THEN
    	timer(DIR:= OUT, TR := SEL(OUT, TOFF, TRUN), RMP := val);
    ELSE
    	val := 255;
    END_IF

    (* when timer = 0 or TEST then initiate autorun until timer reaches 255 *)
    IF (NOT ARX AND ARE AND val = 0) OR TEST THEN
    	val := 0;
    	ARO := TRUE;
    	ARX := TRUE;
    ELSIF val = 255 AND ARO THEN
    	ARO := FALSE;
    	ARX := FALSE;
    END_IF

    (* output is true when autorun ARO is true or IN = TRUE *)
    OUT := IN OR ARO;

    (* revision history
    hm 20. nov. 2008	rev 1.0
    	original version

    *)
END_FUNCTION_BLOCK

(* ---- BLIND_ACTUATOR.st ---- *)
FUNCTION_BLOCK BLIND_ACTUATOR
    (*http://www.oscat.de/images/OSCATBuilding/oscat_building100_en.pdf#page=74*)
    (* make sure only one motor is active at a given time *)
    lock(i1 := UP, I2 := DN, TL := T_LOCKOUT);

    (* ramp UP or down to simulate the angle position of the blind slats *)
    angle(e := lock.Q1 OR lock.Q2, UP := lock.Q1, PT := T_ANGLE);
    position(e := lock.Q1 AND angle.high OR lock.Q2 AND angle.low, UP := lock.Q1, PT := T_UD);

    (* set the outputs *)
    POS := position.Out;
    ANG := angle.Out;

    (* set the outputs *)
    QU := lock.Q1;
    QD := lock.Q2;

    (* set the STATUS output *)
    IF UP AND DN THEN
    	 STATUS := 1;			(* error UP and down together are not allowed *)
    ELSIF UP THEN
    	STATUS := 121;
    ELSIF DN THEN
    	STATUS := 122;
    ELSE
    	STATUS := S_IN;
    END_IF

    (* revision history
    hm	29. sep 2007	rev 1.0
    	original release

    hm	6. oct 2007	rev 1.1
    	rearanged outputs

    hm	18. oct. 2008	rev 1.2
    	changed calls for rmp_B because of change in RMP_B

    hm	27. jul. 2009	rev 1.3
    	changes STATUS to be 12X

    ae	08. mar. 2010 rev 1.4
    	at aPosition

    *)
END_FUNCTION_BLOCK

(* ---- BLIND_CONTROL.st ---- *)
FUNCTION_BLOCK BLIND_CONTROL
    (*http://www.oscat.de/images/OSCATBuilding/oscat_building100_en.pdf#page=75*)
    IF bTimeTest THEN
    	PI:=iPos;
    	AI:=iAngel;
    	UP:=TRUE;
    	DN:=TRUE;
    END_IF

    (* Check Position*)
    act(T_UD:=T_UD, T_ANGLE:=T_ANGLE, T_LOCKOUT := T_LOCKOUT);

    IF UP AND DN THEN
    	(* automatic modus detected *)
    	(* first find correct position *)
    	IF BYTE_TO_INT(act.POS) < BYTE_TO_INT(PI) - delta THEN
    		act.UP := TRUE;
    		act.DN := FALSE;
    		delta := 0;
    		STATUS := 121;
    	ELSIF BYTE_TO_INT(act.POS) > BYTE_TO_INT(PI) + delta THEN
    		act.UP := FALSE;
    		act.DN := TRUE;
    		delta := 0;
    		STATUS := 122;
    	(* regulate angle *)
    	ELSIF BYTE_TO_INT(act.ANG) < BYTE_TO_INT(AI) - delta AND T_ANGLE > T#100ms THEN
    		act.UP := TRUE;
    		act.DN := FALSE;
    		delta := SENS/2;
    		STATUS := 123;
    	ELSIF BYTE_TO_INT(act.ANG) > BYTE_TO_INT(AI) + delta AND T_ANGLE > T#100ms THEN
    		act.UP := FALSE;
    		act.DN := TRUE;
    		delta := SENS/2;
    		STATUS := 124;
    	(* correct position reached *)
    	ELSE
    		act.UP := FALSE;
    		act.DN := FALSE;
    		delta := SENS;
    		STATUS := S_IN;
    	END_IF
    ELSE
    	act.UP := UP;
    	act.DN := DN;
    	STATUS := S_IN;
    END_IF

    (* blind control calls blind_actuator *)
    act(T_UD:=T_UD, T_ANGLE:=T_ANGLE, T_LOCKOUT := T_LOCKOUT);
    POS := act.POS;
    ANG := act.ANG;
    MU := act.QU;
    MD := act.QD;
    STATUS := act.STATUS;

    (* revision history
    hm	29. sep 2007	rev 1.0
    	original release

    hm	6. oct 2007	rev 1.1
    	rearranged outputs
    	integrated blind_actuator into blind_control

    hm	16. oct 2007	rev 1.2
    	ignore angle when T_ANGLE = 0

    hm 29. oct 2007	rev 1.3
    	added lockout configuration time for motor direction change
    	SENS has a setup value of 5

    hm	27. jul. 2009	rev 1.4
    	changed STATUS handling

    ae	08. mar. 2010	rev 1.5
    	at aPosition bevor control
    	at tolerance "delta := SENS/2;"

    *)
END_FUNCTION_BLOCK

(* ---- BLIND_CONTROL_S.st ---- *)
FUNCTION_BLOCK BLIND_CONTROL_S
    (*http://www.oscat.de/images/OSCATBuilding/oscat_building100_en.pdf#page=78*)

    (* STATUS definition
    	121 = manual UP				manual UP operation UP = true and DN = false
    	122 = manual down			manual down operation DN = true and UP = false
    	123 = auto positioning		automatic mode DN = UP = TRUE
    	124 = revert					revert from top or bottom
    	125 = nothing					default input for S_IN
    	127 = Lockout time			lockout between directional change
    	128 = calibrate				calibrate after power UP
    	129 = extend					extend runtime at top or bottom for continuous calibration
    *)

    (* read system time *)
    tx := DWORD_TO_TIME(T_PLC_MS());

    (* check inputs and start state machine *)
    IF UP  AND NOT DN THEN
    	(*  manual UP *)
    	rmp.IN := 255;
    	STATUS := 121;
    ELSIF DN AND NOT UP THEN
    	(* manual DN *)
    	rmp.IN := 0;
    	STATUS := 122;
    ELSIF NOT (UP OR DN) THEN
    	(* manual standby mode *)
    	rmp.IN := PI;
    	STATUS := S_IN;
    END_IF

    (* simulate POS output *)
    rmp(E := UP OR DN, TR := T_UP, TF := T_DN, TL := T_LOCKOUT, OUT := POS);

    (* state machine *)
    CASE STATUS OF
    	0:		(* power UP init *)
    		last := tx;
    		PI_last := PI XOR BYTE#255;
    		STATUS := 128;		(* calibrate *)

    	121: 	(* manual UP *)
    		MU := TRUE;
    		MD := FALSE;
    		IF POS >= (BYTE#255 - EXT_TRIG) THEN
    			(* extend cycle if top is reached *)
    			POS := 255;
    			last := tx;
    			STATUS := 129;	(* extend *)
    		END_IF

    	122:	(* manual down *)
    		MD := TRUE;
    		MU := FALSE;
    		IF POS <= EXT_TRIG THEN
    			(* extend cycle if bottom is reached *)
    			POS := 0;
    			last := tx;
    			STATUS := 129;	(* extend *)
    		END_IF

    	123:	(* auto positioning *)
    		MD := rmp.DN;
    		MU := rmp.UP;
    		IF NOT (rmp.DN OR rmp.UP) THEN
    			(* automatic position is reached *)
    			IF POS <= EXT_TRIG THEN
    				(* extend at bottom *)
    				MD := TRUE;
    				last := tx;
    				STATUS := 129;	(* extend *)
    			ELSIF POS >= (BYTE#255 - EXT_TRIG)  THEN
    				(* extend at top *)
    				MU := TRUE;
    				last := tx;
    				STATUS := 129;	(* extend *)
    			ELSE
    				STATUS := S_IN;
    			END_IF
    		END_IF

    	124:	(* revert from top or bottom *)
    		MD := rmp.DN;
    		MU := rmp.UP;
    		IF NOT(rmp.DN OR rmp.UP) THEN
    (*		IF POS = rmp.IN THEN  *)
    			PI_last := PI;
    			STATUS := S_IN;
    		END_IF

    	127:	(* lockout time *)
    		IF (tx - last) >= T_LOCKOUT THEN
    				STATUS := S_IN;
    		END_IF

    	128:	(* calibration *)
    		MU := TRUE;
    		MD := FALSE;
    		rmp.IN := 255;
    		IF (tx - last) >= (T_UP +  T_EXT) THEN
    			MU := FALSE;
    			last := tx;
    			STATUS := 127;	(* lockout *)
    		END_IF

    	129: (* extend mode *)
    		IF (tx - last) >= T_EXT THEN
    			MU := FALSE;
    			MD := FALSE;
    			last := tx;
    			STATUS := 127;	(* lockout *)
    		END_IF

    ELSE
    	MU := FALSE;
    	MD := FALSE;
    	IF PI <> PI_last THEN
    		PI_last := PI;
    		rmp.IN := PI;
    		STATUS := 123;	(* auto positioning *)
    	ELSIF POS = 0 AND RU THEN
    		rmp.IN := R_POS_BOT;
    		STATUS := 124;	(* revert *)
    	ELSIF POS = 255 AND RD THEN
    		rmp.IN := R_POS_TOP;
    		STATUS := 124;	(* revert *)
    	ELSE
    		STATUS := S_IN;
    	END_IF
    END_CASE

    (* revision history

    hm	9. mar. 2009	rev 1.0
    	original release

    hf	27. jul 2009	rev 1.1
    	major code changes and updates

    hf	23. Jan 2010	rev 1.2
    	fixed a bug during calibration
    	added T_UP and T_DN

    *)
END_FUNCTION_BLOCK

(* ---- BLIND_INPUT.st ---- *)
FUNCTION_BLOCK BLIND_INPUT
    (*http://www.oscat.de/images/OSCATBuilding/oscat_building100_en.pdf#page=80*)
    (* read system timer *)
    tx := DWORD_TO_TIME(T_PLC_MS());

    (* inputs S1 and S2 are debounced and then decoded for multiple clicks *)
    s1e(IN := S1, pt := DEBOUNCE_TIME);
    s2e(IN := S2, pt := DEBOUNCE_TIME);
    s1d(IN := (s1e.Q AND NOT SINGLE_SWITCH) OR (s1e.Q AND SINGLE_SWITCH AND dir), t_long := CLICK_TIME);
    s2d(IN := (s2e.Q AND NOT SINGLE_SWITCH) OR (s1e.Q AND SINGLE_SWITCH AND NOT dir), t_long := CLICK_TIME);

    (* if D1 and D2 are not toggle clear them to make sure they are only active for oine cycle *)
    IF NOT D1_TOGGLE THEN D1 := FALSE; END_IF
    IF NOT D2_TOGGLE THEN D2 := FALSE; END_IF

    (* decode actions *)
    IF (s1d.LONG AND s2d.LONG) OR (STATUS = 139) THEN
       STATUS := 139;
       IF NOT (s1d.LONG OR s2d.LONG)  THEN STATUS := 130; END_IF
    ELSIF s1d.tp_LONG THEN
    	STATUS := 132;
    ELSIF s2d.tp_LONG THEN
    	STATUS := 133;
    ELSIF  s1d.SINGLE THEN
    	IF CLICK_EN THEN
    		(* if running then we stop otherwise start new direction *)
    		IF QU XOR QD THEN
    			STATUS := 131;
    		ELSE
    			STATUS := 134;
    			last := tx;
    			dir := NOT dir;
    		END_IF
    	END_IF
    ELSIF  s2d.SINGLE THEN
    	IF CLICK_EN THEN
    		(* if running then we stop otherwise start new direction *)
    		IF QU XOR QD THEN
    			STATUS := 131;
    		ELSE
    			STATUS := 135;
    			last := tx;
    			dir := NOT dir;
    		END_IF
    	END_IF
    ELSIF IN THEN
    	STATUS := 136;
    	last := tx;
    ELSIF s1d.DOUBLE THEN
    	IF DBL_CLK1 THEN
    		(* a position need to be set for a double click on S1 *)
    		STATUS := 137;
    		last := tx;
    	ELSE
    		(* toggle the output when DBL_CLK1 is not active *)
    		D1 := NOT D1;
    	END_IF
    ELSIF s2d.DOUBLE THEN
    	IF DBL_CLK2 THEN
    		(* a position need to be set for a double click on S2 *)
    		STATUS := 138;
    		last := tx;
    	ELSE
    		(* toggle the output when DBL_CLK2 is not active *)
    		(* IN single switch mode we need to toggle D1 instead of D2 *)
    		IF SINGLE_SWITCH THEN D1 := NOT D1; ELSE D2 := NOT D2; END_IF
    	END_IF
    END_IF

    (* state machine *)
    CASE STATUS OF
    	0:		(* power up operation *)
    			STATUS := 130;

    	130:	(* automatic operation standby *)
    			IF NOT MASTER_MODE THEN
    				PO := POS;
    				AO := ANG;
    			END_IF
    			QU := TRUE;
    			QD := TRUE;

    	131:	(* manual operation standby *)
    			QU := FALSE;
    			QD := FALSE;
    			PO := POS;
    			AO := ANG;
    			(* manual mode will be ended when timeout is reached *)
    			IF tx - last >= MANUAL_TIMEOUT THEN
    				STATUS := 130;
    			END_IF

    	132:	(* manual operation up *)
    			QU := TRUE;
    			QD := FALSE;
    			PO := POS; AO := ANG;
    			last := tx;
    			IF NOT s1d.LONG THEN STATUS := 131; dir := NOT dir; END_IF

    	133:	(* manual operation down *)
    			QU := FALSE;
    			QD := TRUE;
    			PO := POS; AO := ANG;
    			last := tx;
    			IF NOT s2d.LONG THEN	STATUS := 131; dir := NOT dir; END_IF

    	134:	(* manual operation single click up *)
    			QU := TRUE;
    			QD := FALSE;
    			PO := POS; AO := ANG;
    			IF tx - last >= MAX_RUNTIME THEN STATUS := 131; END_IF

    	135:	(* manual operation single click dn *)
    			QU := FALSE;
    			QD := TRUE;
    			PO := POS; AO := ANG;
    			IF tx - last >= MAX_RUNTIME THEN STATUS := 131;	END_IF

    	136:	(* forced input IN = true *)
    			QU := TRUE;
    			QD := TRUE;
    			PO := PI; AO := AI;
    			IF tx-last >= MAX_RUNTIME THEN STATUS := 130; END_IF

    	137:	(* double click1 position *)
    			QU := TRUE;
    			QD := TRUE;
    			PO := DBL_POS1;
    			AO := DBL_ANG1;
    			IF tx - last >= MAX_RUNTIME THEN STATUS := 131; END_IF

    	138:	(* double click2 position *)
    			QU := TRUE;
    			QD := TRUE;
    			PO := DBL_POS2;
    			AO := DBL_ANG2;
    			IF tx - last >= MAX_RUNTIME THEN STATUS := 131; END_IF

    	   139:   (* manual operation standby *)
    	         QU := FALSE;
    	         QD := FALSE;
    	         PO := POS;
    	         AO := ANG;

    END_CASE

    (* revision history
    hm	29. sep 2007	rev 1.0
    	original release

    hm	6. oct 2007		rev 1.1
    	renamed ps and as to PO and AO

    hm	30. dec 2007	rev 1.2
    	added click_timeout variable and function

    hm	16. jul. 2008	rev 1.3
    	rewirtten code to allow for more functionality
    	added single click mode with SINGLE_SWITCH.
    	added Debounce for inputs S1 and S2
    	added double_click functionality

    hm	26. sep. 2008	rev 1.4
    	corrected an error while POS and ANG was transferred to outputs PO and AO during automatic modes

    hm	22. jan 2009	rev 1.5
    	added pulse mode for double click outputs
    	added automatic mode for IN

    hm	27. jul 2009	rev 1.6
    	changed STATUS 0 to 130

    HF	12. nov. 2009	rev 1.7
    	added state 139
    	set defaults for QU, QD, PO

    *)
END_FUNCTION_BLOCK

(* ---- BLIND_NIGHT.st ---- *)
FUNCTION_BLOCK BLIND_NIGHT
    (*http://www.oscat.de/images/OSCATBuilding/oscat_building100_en.pdf#page=84*)
    IF NOT (UP AND DN) AND night THEN
    	(* manual operation at night will cancel operation for one night *)
    	night := FALSE;
    ELSIF (DT_TO_TOD(DTIN) > SUNSET + SUNSET_OFFSET) AND (last_night < DT_TO_DATE(DTIN)) AND NOT night AND E_NIGHT THEN
    	(* enable night *)
    	night := TRUE;
    	last_night := DT_TO_DATE(DTIN);
    ELSIF (DT_TO_TOD(DTIN) > SUNRISE + SUNRISE_OFFSET) AND (last_day < DT_TO_DATE(DTIN)) AND night AND E_DAY AND (last_night < DT_TO_DATE(DTIN)) THEN
    	(* disable night *)
    	night := FALSE;
    	last_day := DT_TO_DATE(DTIN);
    END_IF

    (* shade at night only in auto mode and enable = true *)
    IF UP AND DN AND night THEN
    	STATUS := 141;
    	PO := NIGHT_POSITION;
    	AO := NIGHT_ANGLE;
    ELSE
    	QU := UP;
    	QD := DN;
    	PO := PI;
    	AO := AI;
    	STATUS := S_IN;
    END_IF

    (* revision history
    hm	29. sep 2007	rev 1.0
    	original version

    hm	5. oct 2007		rev 1.1
    	added enable input

    hm	6. oct 2007		rev 1.2
    	added pos and angle inputs and outputs
    	night position and angle can now be configured
    	any manual operation at night will cancel night operation

    *)
END_FUNCTION_BLOCK

(* ---- BLIND_SCENE.st ---- *)
FUNCTION_BLOCK BLIND_SCENE
    (*http://www.oscat.de/images/OSCATBuilding/oscat_building100_en.pdf#page=87*)
    (* delete all bits except the lower 4 of SCENE *)
    x := SCENE AND 16#0F;

    IF ENABLE AND sx[x,2] > 0 AND UP AND DN THEN
    	PO := sx[x,0];
    	AO := sx[x,1];
    	STATUS := 160 + x;  (* STATUS number is 160 to 175 for the 16 scenes *)
    	QU := TRUE;
    	QD := TRUE;
    ELSE
    	QU := UP;
    	QD := DN;
    	STATUS := S_IN;
    	PO := PI;
    	AO := AI;
    END_IF

    (* write SCENE if necessary *)
    IF SWRITE THEN
    	STATUS := 176;		(* write SCENE *)
    	sx[x,0] := PI;
    	sx[x,1] := AI;
    	IF ENABLE THEN sx[x,2] := 1; ELSE sx[x,2] := 0; END_IF (* if sx[x,2] = 0 the SCENE is disabled *)
    END_IF

    (* revision history
    hm	24. oct 2007	rev 1.0
    	original release

    hm		29.1.2008	rev 1.1
    	replaced shr/shl with and for better performance
    *)

END_FUNCTION_BLOCK

(* ---- BLIND_SECURITY.st ---- *)
FUNCTION_BLOCK BLIND_SECURITY
    (*http://www.oscat.de/images/OSCATBuilding/oscat_building100_en.pdf#page=89*)
    IF FIRE THEN
    	QU := TRUE;
    	QD := FALSE;
    	STATUS := 111;
    ELSIF WIND THEN
    	QU := WIND_UP;
    	QD := NOT WIND_UP;
    	STATUS := 112;
    ELSIF ALARM THEN
    	QU := ALARM_UP;
    	QD := NOT ALARM_UP;
    	STATUS := 113;
    ELSIF DOOR THEN
    	QU := TRUE;
    	QD := FALSE;
    	STATUS := 114;
    ELSIF RAIN AND NOT (UP XOR DN) THEN
    	QU := RAIN_UP;
    	QD := NOT RAIN_UP;
    	STATUS := 115;
    ELSE
    	QU := UP;
    	QD := DN;
    	STATUS := S_IN;
    	PO := PI;
    	AO := AI;
    END_IF

    (* revision history
    hm	29. sep 2007	rev 1.0
    	original release

    hm	6. oct 2007		rev 1.1
    	added pos and angle inputs and outputs
    	manual will override RAIN position
    	ALARM position can now be configured

    hm		12. feb. 2008	rev 1.2
    	added config variables RAIN_UP and WIND_UP
    	position for RAIN and WIND is now configurable
    *)

END_FUNCTION_BLOCK

(* ---- BLIND_SET.st ---- *)
FUNCTION_BLOCK BLIND_SET
    (*http://www.oscat.de/images/OSCATBuilding/oscat_building100_en.pdf#page=91*)
    (* read system time *)
    tx := DWORD_TO_TIME(T_PLC_MS());

    (* check inputs *)
    IF IN THEN
    	IF OVERRIDE_MANUAL OR (UP AND DN) THEN
    		STATUS := 178;
    	END_IF
    END_IF

    (* state machine *)
    CASE STATUS OF
    	0: (* power on state *)
    		STATUS := S_IN;

    	178: (* force values from PX and AX *)
    		PO := PX;
    		AO := AX;
    		QU := TRUE;
    		QD := TRUE;
    		(* check for end of forced position *)
    		IF NOT IN THEN
    			STATUS := SEL(RESTORE_POSITION, S_IN, 179);
    			last := tx;
    		END_IF

    	179: (* restore previous position *)
    		PO := ps;
    		AO := as;
    		IF ((PO = PI) AND (AO = AI))  OR tx - last >= RESTORE_TIME THEN
    			STATUS := S_IN;
    		END_IF

    ELSE
    	(* no operation transfer inputs to outputs *)
    	PO := PI;
    	ps := PI;
    	AO := AI;
    	as := AI;
    	STATUS := S_IN;
    	QU := UP;
    	QD := DN;
    END_CASE

    (* revision history
    hm	27. jul 2009	rev 1.0
    	original release

    *)
END_FUNCTION_BLOCK

(* ---- BLIND_SHADE.st ---- *)
FUNCTION_BLOCK BLIND_SHADE
    (*http://www.oscat.de/images/OSCATBuilding/oscat_building100_en.pdf#page=93*)
    (* the input SUN is sent through tof which will delay the shade for the time SHADE_DELAY *)
    sun_delay(IN := SUN, PT := SHADE_DELAY);

    IF UP AND DN AND ENABLE AND sun_delay.Q AND CX.SUN_HOR > DIRECTION - ANGLE_OFFSET AND CX.SUN_HOR < DIRECTION + ANGLE_OFFSET AND
    	DT_TO_TOD(CX.UTC) > CX.SUN_RISE + SUNRISE_OFFSET AND DT_TO_TOD(CX.UTC) < CX.SUN_SET - SUNSET_PRESET THEN
    	STATUS := 151;
    	QU := UP;
    	QD := DN;
    	(* position is predefined *)
    	PO := SHADE_POS;
    	(* shading is active now calculate the slat angle *)
    	(* calculate the max angle for the blind *)
    	angle := DEG(ATAN(SLAT_SPACING / SLAT_WIDTH));
    	(* check if SUN angle is between 0 and max angle *)
    	IF CX.SUN_VER > 0.0 AND CX.SUN_VER < angle THEN
    		angle := CX.SUN_VER + DEG(ACOS(COS(RAD(CX.SUN_VER))*SLAT_SPACING / SLAT_WIDTH));
    		AO := INT_TO_BYTE(DINT_TO_INT(LIMIT(0,TRUNC(angle * 2.833333333), 255)));
    	ELSE
    		AO := 255;
    	END_IF
    ELSE
    	QU := UP;
    	QD := DN;
    	PO := PI;
    	AO := AI;
    	STATUS := S_IN;
    END_IF

    (* revision history
    hm	15 oct. 2007	rev 1.0
    	original version

    hm	19. oct 2007	rev 1.1
    	manual mode was not detected because outputs were checked and not inputs UP and DN

    hm	24. nov 2007	rev 1.2
    	added SHADE_DELAY to avoid constant UP and down if SUN is out parcially

    hm	8. feb 2009	rev 1.3
    	added shading position SHADE_POS to be configured
    	changed inputs to utilize calendar data structure

    hm	13. mar. 2009	rev 1.4
    	improved code

    *)
END_FUNCTION_BLOCK

(* ---- BLIND_SHADE_S.st ---- *)
FUNCTION_BLOCK BLIND_SHADE_S
    (*http://www.oscat.de/images/OSCATBuilding/oscat_building100_en.pdf#page=96*)
    (* STATUS definition
       151 = shadow               move shutter down for shadowing
       152 = ALERT                  move shutter UP by setting QU:=TRUE when door is open.
    *)

    (* the input SUN is sent through tof which will delay the shade for the time SHADE_DELAY *)
    sun_delay(IN := SUN, PT := SHADE_DELAY);

    IF ALERT THEN
       QU := TRUE;
       QD := FALSE;
       STATUS := 152;
    ELSIF UP AND DN AND ENABLE AND sun_delay.Q
    AND (CX.SUN_HOR > HORZ1) AND (CX.SUN_HOR < HORZ2)
    AND (CX.SUN_VER < VERT)
    AND (DT_TO_TOD(CX.UTC) > CX.SUN_RISE + SUNRISE_OFFSET) AND (DT_TO_TOD(CX.UTC) < CX.SUN_SET - SUNSET_PRESET) THEN
       QU := UP;
       QD := DN;
       STATUS := 151;
       (* Calculate Position, must be SHADE_POS or less *)
       PO := MIN(PI, SHADE_POS);
    ELSE
       QU := UP;
       QD := DN;
       PO := PI;
       STATUS := S_IN;
    END_IF

    (* revision history
    hf	12 nov. 2009	rev 1.0
    	original version

    *)
END_FUNCTION_BLOCK

(* ---- BOILER.st ---- *)
FUNCTION_BLOCK BOILER
    (*http://www.oscat.de/images/OSCATBasic/oscat_basic333_en.pdf#page=428*)
    (* read sensors and check for valid data *)
    IF T_UPPER > T_PROTECT_HIGH THEN
    	STATUS := 1;
    	HEAT := FALSE;
    	ERROR := TRUE;
    ELSIF T_UPPER < T_PROTECT_LOW THEN
    	STATUS := 2;
    	HEAT :=	TRUE;
    	ERROR := TRUE;
    ELSIF T_LOWER > T_PROTECT_HIGH AND T_LOWER_ENABLE THEN
    	STATUS := 3;
    	HEAT := FALSE;
    	ERROR := TRUE;
    ELSIF T_LOWER < T_PROTECT_LOW AND T_LOWER_ENABLE THEN
    	STATUS := 4;
    	HEAT := TRUE;
    	ERROR := TRUE;
    ELSIF NOT PRESSURE THEN
    	STATUS := 5;
    	HEAT := FALSE;
    	ERROR := TRUE;
    ELSIF REQ_1 OR REQ_2 OR ENABLE OR BOOST THEN
    	ERROR := FALSE;

    	(* determine if HEAT needs to be turned on *)
    	IF BOOST AND NOT edge_ AND T_UPPER < T_UPPER_MAX THEN
    		STATUS := 101;
    		HEAT := TRUE;
    		boost_mode := TRUE;
    	ELSIF ENABLE AND T_UPPER < T_UPPER_MIN THEN
    		STATUS := 102;
    		HEAT := TRUE;
    	ELSIF REQ_1 AND T_UPPER < T_REQUEST_1 THEN
    		STATUS := 103;
    		HEAT := TRUE;
    	ELSIF REQ_2 AND T_UPPER < T_REQUEST_2 THEN
    		STATUS := 104;
    		HEAT := TRUE;
    	END_IF

    	(* determine the shut off temperature *)
    	IF HEAT THEN
    		IF (ENABLE OR boost_mode) THEN
    			flag_0 := TRUE;
    			IF T_LOWER_ENABLE AND T_LOWER > T_LOWER_MAX THEN
    				flag_0 := boost_mode := FALSE;
    			ELSIF NOT T_LOWER_ENABLE AND T_UPPER > T_UPPER_MAX THEN
    				flag_0 := boost_mode := FALSE;
    			END_IF
    		ELSE
    			flag_0 := FALSE;
    		END_IF
    		flag_1 := (REQ_1 AND T_UPPER > T_REQUEST_1 + T_REQUEST_HYS) AND REQ_1;
    		flag_2 := (REQ_2 AND T_UPPER > T_REQUEST_2 + T_REQUEST_HYS) AND REQ_2;

    		(* shut off HEAT if no longer needed *)
    		HEAT := flag_0 OR flag_1 OR flag_2;
    		IF HEAT = FALSE THEN STATUS := 100; END_IF
    	END_IF
    ELSE
    	STATUS := 100;
    	HEAT := FALSE;
    	ERROR := FALSE;
    END_IF
    edge_ := BOOST;

    (* revision history
    hm	27. feb. 2007	rev 1.0
    	original version

    hm	16. oct. 2008	rev 1.1
    	improved performance

    hm	13. mar. 2009	rev 1.2
    	real constants updated to new systax using dot
    	replaced double assignments
    *)
END_FUNCTION_BLOCK

(* ---- BURNER.st ---- *)
FUNCTION_BLOCK BURNER
    (*http://www.oscat.de/images/OSCATBasic/oscat_basic333_en.pdf#page=430*)
    (* read system time *)
    tx := DWORD_TO_TIME(T_PLC_MS());

    (* check RST input and overtemp *)
    IF RST OR OVER_TEMP OR state = 0 THEN
    	IF STATUS > 0 AND tx - last_change >= LOCKOUT_TIME AND RST THEN
    		STATUS := 110;
    		FAIL := FALSE;
    		state := 1;
    	ELSE
    		(* normaler reset *)
    		MOTOR := FALSE;
    		COIL1 := FALSE;
    		COIL2 := FALSE;
    		IGNITE := FALSE;
    		PRE_HEAT := FALSE;
    		IF OVER_TEMP THEN
    			STATUS := 9;
    			FAIL := TRUE;
    		END_IF
    		last_change := tx;
    		last := tx;
    		state := 1;
    	END_IF
    END_IF

    (* check for timer RST and RST timer if true *)
    IF RST_TIMER THEN
    	RUNTIME1 := 0;
    	RUNTIME2 := 0;
    	CYCLES := 0;
    	cycles2 := 0;
    END_IF

    (* quit here if an error is present *)
    IF (STATUS > 0 AND STATUS < 100) OR RST THEN RETURN; END_IF

    (* start sequence *)
    CASE state OF

    1:	(* IN signal starts oil pre heating *)
    	IF IN AND FLAME THEN
    		state := 7;
    		PRE_HEAT := FALSE;
    		STATUS := 2;
    		last_change := tx;
    	ELSIF IN THEN
    		PRE_HEAT := TRUE;
    		state := 2;
    		last_change := tx;
    	END_IF

    2:	(* after pre_heating time start MOTOR *)
    	IF (tx- last_change >= PRE_HEAT_TIME AND OIL_TEMP) OR (OIL_TEMP AND NOT oil_temp_last) THEN
    		MOTOR := TRUE;
    		state := 3;
    		last_change := tx;
    	(* PRE_HEAT_TIME ist abgelaufen und OIL_TEMP ist nicht aktiv *)
    	ELSIF tx - last_change >= PRE_HEAT_TIME AND NOT OIL_TEMP THEN
    		state := 7;
    		PRE_HEAT := FALSE;
    		STATUS := 1;
    		last_change := tx;
    	(* FLAME monitor cannot be active at this time *)
    	ELSIF FLAME THEN
    		state := 7;
    		PRE_HEAT := FALSE;
    		STATUS := 2;
    		last_change := tx;
    	END_IF

    3:	(* abwarten bis zündung eingeschaltet werden kann *)
    	IF tx - last_change >= PRE_VENT_TIME - PRE_IGNITE_TIME THEN
    		IGNITE := TRUE;
    		state := 4;
    		last_change := tx;
    	(* FLAME monitor cannot be active at this time *)
    	ELSIF FLAME THEN
    		state := 7;
    		PRE_HEAT := FALSE;
    		MOTOR := FALSE;
    		STATUS := 3;
    		last_change := tx;
    	END_IF

    4:	(* warten bis oelzufuhr geoeffnet werden darf *)
    	IF tx - last_change >= PRE_IGNITE_TIME THEN
    		COIL1 := TRUE;
    		state := 5;
    		last_change := tx;
    	END_IF

    5:	(* warten auf flammwaechter und falls noetig abschalten *)
    	IF tx - last_change >= SAFETY_TIME OR FLAME THEN
    		IF NOT FLAME THEN
    			(* notabschaltung da flammwaechster nicht angesprochen hat *)
    			state := 7;
    			MOTOR := FALSE;
    			COIL1 := FALSE;
    			PRE_HEAT := FALSE;
    			IGNITE := FALSE;
    			STATUS := 4;
    			last_change := tx;
    		ELSE
    			state := 6;
    			last_change := tx;
    		END_IF
    	END_IF

    6:	(* brenner läuft, flammueberwachung und nach ablauf der nachigniteszeit IGNITE abschalten *)
    	IF NOT FLAME AND NOT MULTIPLE_IGNITION THEN
    		(* notabschaltung da flammwaechster keine flamme meldet *)
    		state := 7;
    		MOTOR := FALSE;
    		COIL1 := FALSE;
    		COIL2 := FALSE;
    		PRE_HEAT := FALSE;
    		IGNITE := FALSE;
    		STATUS := 5;
    		last_change := tx;
    	ELSIF NOT FLAME AND MULTIPLE_IGNITION THEN
    		IGNITE := TRUE;
    		state := 5;
    		COIL2 := FALSE;
    		last_change := tx;
    	ELSE
    		IF tx - last_change >= POST_IGNITE_TIME THEN
    			(* POST_IGNITE_TIME abgelaufen, IGNITE abschalten *)
    			IGNITE := FALSE;
    		END_IF
    		IF tx - last_change >= STAGE2_DELAY AND STAGE2 THEN
    			COIL2 := TRUE;
    		ELSE
    			COIL2 := FALSE;
    		END_IF
    	END_IF
    END_CASE

    (* abschaltung wenn kein eingangssignal *)
    IF NOT IN THEN
    	state := 1;
    	MOTOR := FALSE;
    	COIL1 := FALSE;
    	COIL2 := FALSE;
    	IGNITE := FALSE;
    	PRE_HEAT := FALSE;
    	last_change := tx;
    END_IF

    (* runtimezähler *)
    timer1(IN := FLAME AND IN AND MOTOR AND COIL1 AND NOT COIL2, seconds := RUNTIME1, CYCLES := CYCLES);
    timer2(IN := FLAME AND IN AND MOTOR AND COIL1 AND COIL2, seconds := RUNTIME2, CYCLES := cycles2);
    KWH := UDINT_TO_REAL(RUNTIME1) * KW1 / 3600.0 + UDINT_TO_REAL(RUNTIME2) * KW2 / 3600.0;

    (* zeit fuer naechsten aufruf merken *)
    last := tx;

    (* set FAIL output IF ERROR and STATUS  if normal operation *)

    IF STATUS > 0 AND STATUS < 100 THEN
    	FAIL := TRUE;
    ELSE
    	FAIL := FALSE;
    	IF NOT IN THEN
    		STATUS := 110;
    	ELSIF FLAME AND IN AND MOTOR AND COIL2 AND COIL1 THEN
    		STATUS := 113;
    	ELSIF FLAME AND IN AND MOTOR AND COIL1 THEN
    		STATUS := 112;
    	ELSE
    		STATUS := 111;
    	END_IF
    END_IF

    (*
    31.12.2006	hm		rev 1.1
    	added PRE_HEAT timing and output
    	FLAME monitor before ignition will generate error on STATUS output
    	added output for KWH

    31.12.2006	hm		rev 1.2
    	added oil_temp_input

    31.12.2006	hm		rev 1.3
    	changed STATUS output to be byte instead of bool

    22.1.2007		hm		rev 1.4
    	renamed FAIL output to STATUS
    	added output CYCLES
    	corrected an error while PRE_HEAT would be on when an error was present
    	added COIL2 output and STAGE2 input

    15.9.2007		hm		rev 1.5
    	replaced Time() with T_PLC_MS for compatibility and performance reasons

    hm	21. oct. 2008	rev 1.6
    	changed code to use new ontime rev 2.0
    *)
END_FUNCTION_BLOCK

(* ---- CLICK.st ---- *)
FUNCTION_BLOCK CLICK
    (*http://www.oscat.de/images/OSCATBuilding/oscat_building100_en.pdf#page=47*)
    (* reconfiguration and debounce circuitry *)
    s_in(IN := IN, TD := T_DEBOUNCE, TR := T_RECONFIG);

    (* read system time *)
    tx := DWORD_TO_TIME(T_PLC_MS());

    (* count the mumber of clicks *)
    IF s_in.Q XOR Q THEN
    	last := tx;
    	IF s_in.Q THEN state := state + 1; END_IF
    END_IF
    Q := s_in.Q;

    (* set outputs *)
    IF state > 0 THEN
    	IF (Q AND tx - last > T_SHORT) OR (NOT Q AND tx - last > T_PAUSE) THEN
    		CASE state OF
    			1:	SINGLE := TRUE;
    				STATUS := 111;
    			2:	DOUBLE := TRUE;
    				STATUS := 112;
    			3:	TRIPLE := TRUE;
    				STATUS := 113;
    		END_CASE
    		state := 0;
    	END_IF
    ELSIF NOT Q THEN
    	SINGLE := FALSE;
    	DOUBLE := FALSE;
    	TRIPLE := FALSE;
    	STATUS := 110;
    	last := tx;
    	state := 0;
    END_IF

    (* revision history

    15 Feb 2007	rev 1.0	hm
    	created original version

    18.5.2007	rev 1.1 hm
    	corrected an error while execution would stop after T_RECONFIG elapsed.

    15.9.2007	rev 1.2 hm
    	replaced Time() with T_PLC_MS for compatibility and performance reasons

    28. dec. 2008	rev 2.0
    	rewritten using modular approach

    *)
END_FUNCTION_BLOCK

(* ---- CLICK_MODE.st ---- *)
FUNCTION_BLOCK CLICK_MODE
    (*http://www.oscat.de/images/OSCATBuilding/oscat_building100_en.pdf#page=49*)
    (* when input goes high start the Timer to decode pulses *)
    Timer(IN := IN, PT := T_LONG);
    SINGLE := FALSE;
    DOUBLE := FALSE;

    IF Timer.Q THEN
    	(* decode pulses while the Timer is active *)
    	IF NOT IN AND last THEN	cnt := cnt + 1; END_IF
    ELSE
    	CASE cnt OF
    		1 : SINGLE := TRUE;
    		2 : DOUBLE := TRUE;
    	END_CASE
    	cnt := 0;
    END_IF
    last := IN;
    TP_LONG := NOT Timer.Q AND (NOT LONG) AND IN;
    LONG := NOT Timer.Q AND IN;

    (* revision history

    hm	13. nov. 2008	rev 1.0
    	original release

    *)
END_FUNCTION_BLOCK

(* ---- DEBOUNCE.st ---- *)
FUNCTION_BLOCK DEBOUNCE
    (*http://www.oscat.de/images/OSCATBuilding/oscat_building100_en.pdf#page=49*)

    IF NOT deb.Q AND IN THEN
    	(* rising edge on input detetced a *)
    	Q := TRUE;
    ELSIF NOT PM THEN
    	Q := deb.Q;
    ELSE
    	Q := FALSE;
    END_IF

    (* run debounce timer *)
    deb(IN := IN, PT := TD);

    (*
    hm 22. sep. 2008	rev 1.0
    	original version

    *)
END_FUNCTION_BLOCK

(* ---- DIMM_2.st ---- *)
FUNCTION_BLOCK DIMM_2
    (*http://www.oscat.de/images/OSCATBuilding/oscat_building100_en.pdf#page=50*)
    (* debouncing for inputs I1 and I2 *)
    t1(IN := I1, PT := T_DEBOUNCE);
    t2(IN := I2, PT := T_DEBOUNCE);
    dc1(in := t1.Q, T_LONG := T_DIMM_START);
    dc2(in := t2.Q, T_LONG := T_DIMM_START);

    IF RST THEN
    	IF RST_OUT THEN OUT := 0; END_IF
    	Q := FALSE;
    	D1 := FALSE;
    	D2 := FALSE;
    ELSIF SET THEN
    	OUT := VAL;
    	Q := TRUE;
    ELSIF dc1.SINGLE THEN
    	(* single click on I1 turns the dimmer on *)
    	OUT := LIMIT(MAX(MIN_ON,1), OUT, MAX_ON);
    	Q := TRUE;
    ELSIF dc2.SINGLE THEN
    	(* single click on I2 turns the dimmer off *)
    	Q := FALSE;
    ELSIF dc1.TP_LONG THEN
    	(* continuous on at I1 dimms up *)
    	IF NOT Q THEN
    		OUT := SEL(SOFT_DIMM, LIMIT(MAX(MIN_ON,1), OUT, MAX_ON), 1);
    	END_IF
    	Q := TRUE;
    	dim.DIR := TRUE;
    ELSIF dc2.TP_LONG THEN
    	(* continuous on at I2 dimms down *)
    	dim.DIR := FALSE;
    END_IF

    (* SET the double click output *)
    IF NOT DBL1_TOG THEN D1 := FALSE; END_IF
    IF dc1.DOUBLE THEN
    	IF DBL1_SET THEN
    		OUT := DBL1_POS;
    		Q := TRUE;
    	ELSE
    		D1 := NOT D1;
    	END_IF
    END_IF
    IF NOT DBL2_TOG THEN D2 := FALSE; END_IF
    IF dc2.DOUBLE THEN
    	IF DBL2_SET THEN
    		OUT := DBL2_POS;
    		Q := TRUE;
    	ELSE
    		D2 := NOT D2;
    	END_IF
    END_IF

    (* while dimming is active ramp the output OUT up or down *)
    dim(dir := dc2.LONG, e := dc1.LONG OR dc2.LONG , TR := T_DIMM, rmp := OUT);

    (* turn off output if a value of 0 is reached *)
    IF OUT = 0 THEN Q := FALSE; END_IF

    (* limit the maximum runtime *)
    IF T_ON_MAX > t#0s THEN
    	t3(in := Q, pt := T_ON_MAX);
    	Q := Q XOR t3.Q;
    END_IF

    (* revision history

    hm 22. mar. 2009	rev 1.0
    	original version

    *)
END_FUNCTION_BLOCK

(* ---- DIMM_I.st ---- *)
FUNCTION_BLOCK DIMM_I
    (*http://www.oscat.de/images/OSCATBuilding/oscat_building100_en.pdf#page=52*)
    (* the input is first sent through auto reconfiguration and debouncing *)
    config(IN := IN, TD := T_DEBOUNCE, TR := T_RECONFIG);
    decode(IN := config.Q, T_LONG := T_DIMM_START);

    IF RST THEN
    	IF RST_OUT THEN OUT := 0; END_IF
    	Q := FALSE;
    	dir := OUT > 127;
    ELSIF SET THEN
    	OUT := VAL;
    	Q := TRUE;
    	(* SET direction to up when value < 127 otherwise SET dir down dir is reversed because next action will reverse again *)
    	dir := OUT > 127;
    ELSIF decode.SINGLE THEN
    	(* a single click reverses output Q *)
    	Q := NOT Q;
    	(* when dimmer is turned on we need to limit OUT to min and max limits *)
    	IF Q THEN	OUT := LIMIT(MAX(MIN_ON,1), OUT, MAX_ON);	END_IF
    	(* SET the appropriate direction of dimmer dir is reversed because next action will reverse again *)
    	dir := OUT > 127;
    ELSIF decode.TP_LONG THEN
    	IF NOT Q THEN
    		IF SOFT_DIMM THEN
    			OUT := 1;
    			dir := TRUE;
    		ELSE
    			OUT := LIMIT(MAX(MIN_ON,1), OUT, MAX_ON);
    			dir := OUT < 127;
    		END_IF
    		Q := TRUE;
    	ELSE
    		(* reverse direction with every long click *)
    		dir := NOT dir;
    	END_IF
    END_IF

    (* SET the double click output *)
    IF NOT DBL_TOGGLE THEN DBL := FALSE; END_IF
    IF decode.DOUBLE THEN DBL := NOT DBL; END_IF

    (* while dimming is active ramp the output OUT up or down *)
    dim(dir := dir, e := decode.LONG AND Q, TR := T_DIMM, rmp := OUT);

    (* reverse direction when limits are reached *)
    IF OUT = 0 THEN
    	dir := TRUE;
    ELSIF OUT = 255 THEN
    	dir := FALSE;
    END_IF

    (* limit the maximum runtime *)
    IF T_ON_MAX > t#0s THEN
    	t3(IN := Q, pt := T_ON_MAX);
    	Q := Q XOR t3.Q;
    END_IF

    (* revision history

    hm 22.1.2007		rev 1.1
    	deleted unused structure ramp

    hm 2.feb 2007		rev 1.2
    	changed structure to read time() at the beginning for better time consistency if a higher priorized tak interrupts dimm_i
    	added statements IN case structure for state 1 to allow for short 1 cycle input pulses

    hm 	15.9.2007		rev 1.3
    	replaced Time() with T_PLC_MS for compatibility and performance reasons

    hm	30. sep. 2008	rev 1.4
    	added Input VAL to supply value for SET input
    	added setup parameter init_val

    hm	22. oct. 2008	rev 2.0
    	new code and features

    hm	14. nov. 2008	rev 2.1
    	added SOFT_DIMM feature

    hm	16. nov. 2008	rev 2.2
    	added reset OUT feature

    hm	26. jan. 2009	rev 2.3
    	dimming will also reverse at OUT = 0
    	RST will override SET
    *)
END_FUNCTION_BLOCK

(* ---- F_LAMP.st ---- *)
FUNCTION_BLOCK F_LAMP
    (*http://www.oscat.de/images/OSCATBuilding/oscat_building100_en.pdf#page=54*)
    runtime(in := SWITCH, seconds := ONTIME, CYCLES := CYCLES);

    IF RST THEN
    	ONTIME := 0;
    	CYCLES := 0;
    END_IF
    IF SWITCH THEN
    	IF ONTIME < T_NO_DIMM * 3600 THEN
    		LAMP := 255;
    		STATUS := 111;
    	ELSE
    		LAMP := DIMM;
    		STATUS := 112;
    	END_IF
    ELSE
    	LAMP := 0;
    	STATUS := 110;
    END_IF

    IF ONTIME >= T_MAINTENANCE * 3600 AND T_MAINTENANCE > 0 THEN
    	STATUS := 120;
    END_IF

    (* revision history
    hm	8. feb. 2007	rev 1.1
    	original version

    hm	22. oct. 2008	rev 1.2
    	changed use of ONTIME for ONTIME 2.0
    	ONTIME is now in seconds not hours
    *)

END_FUNCTION_BLOCK

(* ---- HEAT_METER.st ---- *)
FUNCTION_BLOCK HEAT_METER
    (*http://www.oscat.de/images/OSCATBasic/oscat_basic333_en.pdf#page=436*)
    IF RST THEN
    	int1(RST := TRUE);
    	int1.RST := FALSE;
    	C := 0.0;
    	Y := 0.0;
    ELSIF E THEN
    	x := (WATER_DENSITY(SEL(RETURN_METER, TF, TR), FALSE) * (WATER_ENTHALPY(TF) - WATER_ENTHALPY(TR)) * (1.0 - CONTENT) + CP * DENSITY * CONTENT * (TF-TR));
    END_IF

    (* integrate or add consumption *)
    int1(run := NOT PULSE_MODE AND E, in := x * LPH * 2.77777777777E-4);
    IF PULSE_MODE THEN
    	IF NOT edge_ AND E THEN Y := Y + x * LPH; END_IF
    ELSE
    	Y := int1.Out;
    END_IF

    (* store the value of E *)
    edge_ := E;

    (* read system_time *)
    tx := T_PLC_MS();

    (* only init at startup necessary *)
    IF NOT init THEN
    	init := TRUE;
    	last := tx;
    END_IF

    (* calculate the current consumption *)
    IF (tx - last >= TIME_TO_DWORD(AVG_TIME)) AND (AVG_TIME > T#0s) THEN
    	last := tx;
    	C := (Y - y_last) * 3.6E6 / DWORD_TO_REAL(TIME_TO_DWORD(AVG_TIME));
    	y_last := Y;
    END_IF

    (* revision history
    hm	16. nov. 2007	rev 1.0
    	original version

    hm	24. dec. 2007	rev 1.1
    	added config variable RETURN_METER
    	added output C for current consumption

    hm	6. mar. 2008	rev 1.2
    	corrected an error in pulse mode

    hm	16. mar. 2008	rev 1.3
    	added type conversion to avoid warnings under codesys 3.0

    hm	21. oct. 2008	rev 1.4
    	improved code

    hm	6. nov. 2008	rev 1.5
    	changed to FT_INT2 to avoid overrun at hig values

    hm	8. feb. 2009	rev 1.6
    	changes Y to be I/O

    hm	23. mar. 2009	rev 1.7
    	real constants updated to new systax using dot
    	corected error in formula

    hm	27. jul 2009	rev 1.8
    	output C is now calculated in J/h

    hm	13. nov. 2009	rev 1.9
    	output C is now calculated correctly

    hm	23. jan. 2011	rev 1.10
    	corrected an error with PULSE_MODE
    *)

END_FUNCTION_BLOCK

(* ---- HEAT_TEMP.st ---- *)
FUNCTION_BLOCK HEAT_TEMP
    (*http://www.oscat.de/images/OSCATBasic/oscat_basic333_en.pdf#page=33*)
    tr := T_INT + OFFSET;
    tx := (tr - T_EXT) / (T_INT_CONFIG - T_EXT_CONFIG);

    IF T_EXT + H > tr THEN
    	TY := 0.0;
    ELSE
    	TY := LIMIT(TY_MIN, tr + T_DIFF * 0.5 * tx + (TY_CONFIG - T_DIFF * 0.5 - tr) * EXPT(tx, 1.0 / C), TY_MAX);
    END_IF

    TY := MAX(TY, T_REQ);
    HEAT := TY > 0.0;

    (*

    tv=ti+(tvmax-ti)*((ti-tau)/(ti-taumin))(1/n)

    tv aktuelle Vorlauftemp.
    ti Raumtemperatur innen (20°C)
    tau aktuelle Außentemperatur
    taumin minimale Außentemperatur -12°C oder -15°C
    n Heizkörperexponent (meistens 1,33)
    Fußbodenheizung = 1,1
    Wandheizung 1,3

    Normen z. B. DIN 4703, DIN 4725 oder die Literatur, z. B Recknagel Abschnitt 1.3.5.

    *)

    (* revision history
    hm	27. jan. 2008	rev 1.0
    	original version

    hm	26. sep. 2008	rev 1.1
    	moved T_INT from config to Input
    	added config variable H
    	corrected error in formula

    hm	13. mar. 2009	rev 1.2
    	improved code

    *)
END_FUNCTION_BLOCK

(* ---- LEGIONELLA.st ---- *)
FUNCTION_BLOCK LEGIONELLA
    (*http://www.oscat.de/images/OSCATBasic/oscat_basic333_en.pdf#page=443*)
    (* startup initialization *)
    IF NOT init THEN
    	init := TRUE;
    	X1.DAY := SHR(BYTE#128,DAY);
    	X1.start := T_START;
    	x3.low := TEMP_OFFSET + TEMP_SET;
    	x3.high := TEMP_HYS + x3.low;
    	x2.wait0 := T_MAX_HEAT;
    	x2.delay0 := TP_0;
    	x2.delay1 := TP_1;
    	x2.delay2 := TP_2;
    	x2.delay3 := TP_3;
    	x2.delay4 := TP_4;
    	x2.delay5 := TP_5;
    	x2.delay6 := TP_6;
    	x2.delay7 := TP_7;
    	x2.wait1 := T_MAX_RET;
    	x2.wait2 := T_MAX_RET;
    	x2.wait3 := T_MAX_RET;
    	x2.wait4 := T_MAX_RET;
    	x2.wait5 := T_MAX_RET;
    	x2.wait6 := T_MAX_RET;
    	x2.wait7 := T_MAX_RET;
    	x2();
    END_IF

    (* oerational code *)
    X1(DTi := DT_IN);
    IF X1.Q OR MANUAL OR x2.RUN THEN
    	x3(in := TEMP_BOILER);
    	x2.in0 := x3.Q OR x3.win;
    	x2.in1 := TEMP_RETURN >= TEMP_SET;
    	x2.in2 := x2.in1;
    	x2.in3 := x2.in1;
    	x2.in4 := x2.in1;
    	x2.in5 := x2.in1;
    	x2.in6 := x2.in1;
    	x2.in7 := x2.in1;
    	x2.RST := RST;
    	x2(start := X1.Q OR MANUAL);
    	RUN := x2.RUN;
    	PUMP := x2.qx;
    	HEAT := NOT x3.Q AND x2.RUN;
    	VALVE0 := x2.Q0;
    	VALVE1 := x2.Q1;
    	VALVE2 := x2.Q2;
    	VALVE3 := x2.Q3;
    	VALVE4 := x2.Q4;
    	VALVE5 := x2.Q5;
    	VALVE6 := x2.Q6;
    	VALVE7 := x2.Q7;
    	PUMP := x2.qx;
    	STATUS := x2.STATUS;
    ELSE;
    	x2(start :=0);
    	STATUS := x2.STATUS;
    END_IF

    (* revision history

    hm 17.jan 2007	rev 1.1
    	rewritten to st for higher performance
    	changes eeror output to esr compatible STATUS output

    hm	23. 10.2008	rev 1.2
    	update code to use new version of timer_1

    hm	13. mar. 2009	rev 1.3
    	real constants updated to new systax using dot
    	using new module sequence_8
    *)

END_FUNCTION_BLOCK
